Staubli VAL3: sign.pgx

public program sign()
begin
end
